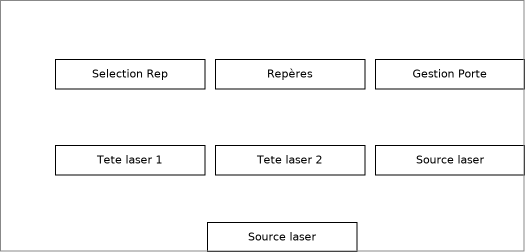
VISUALIZATION MenuPrincipal  // 525x252
    Rectangle (55,59 150x30), "Selection Rep"
        OnMouseClick: change screen: Selection_Rep
    Rectangle (215,59 150x30), "Repères"
        OnMouseClick: change screen: chgt_Reperes
    Rectangle (55,145 150x30), "Tete laser 1"
        OnMouseClick: change screen: Laser_Tete_Raytools_1
    Rectangle (215,145 150x30), "Tete laser 2"
        OnMouseClick: change screen: Laser_Tete_Raytools_2
    Rectangle (375,145 150x30), "Source laser"
        OnMouseClick: change screen: Visualization_source
    Rectangle (375,59 150x30), "Gestion Porte"
        OnMouseClick: change screen: Porte_secu
    Rectangle (207,222 150x30), "Source laser"
        OnMouseClick: change screen: StateEthercat
END_VISUALIZATION

(* stored: Version 1.1.0.1
   Visu MenuPrincipal: Id {bb3e8a36-ef87-4685-874f-3648ac189e4b} *)
